% RSLogix 500 project I2P-Job-12 Part 2 Duncan_Sutton.RSS, saved by version 10.00.00.00 %
PROJECT "ML01A"    % processor: Bul.1763 MicroLogix 1100 Series B %

PROGRAM FILES
  LAD 2   9 rungs

DATA FILES
  O0 OUTPUT  4 elements
  I1 INPUT  6 elements
  S2 STATUS  66 elements
  B3 BINARY  1 elements
  T4 TIMER  1 elements
  C5 COUNTER  1 elements
  R6 CONTROL  1 elements
  N7 INTEGER  1 elements
  F8 FLOAT  1 elements

LADDER 2
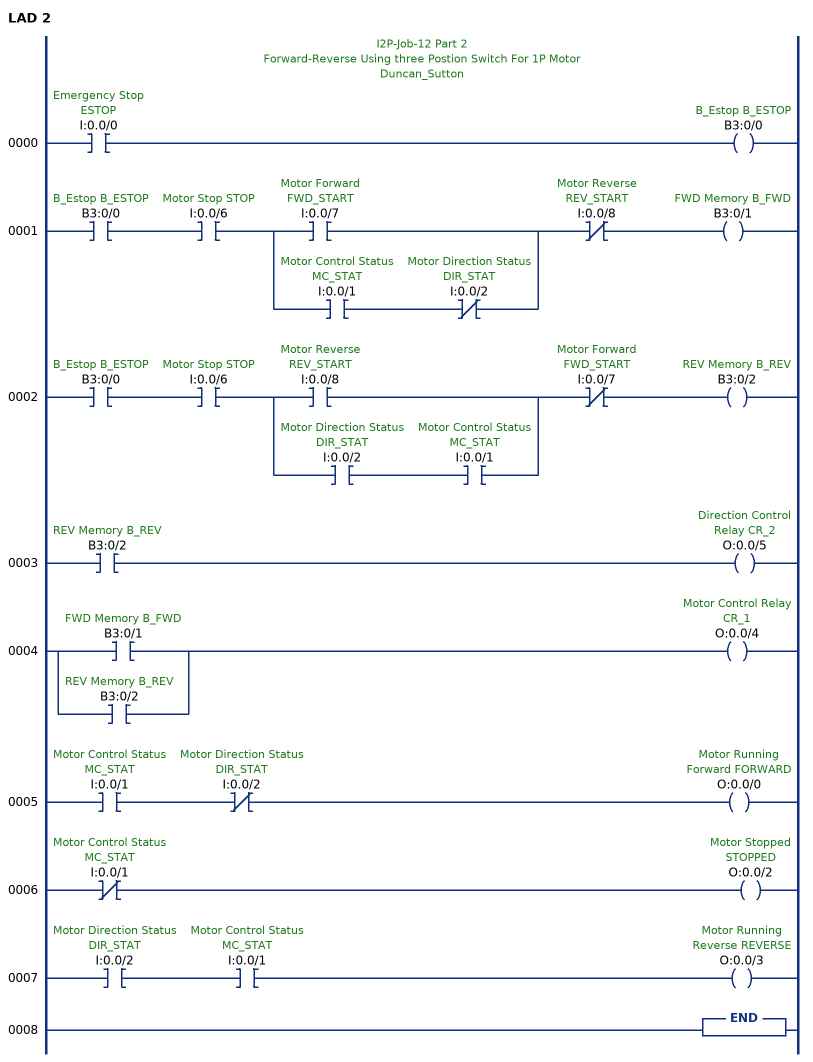
% Rung: 0 %
% I2P-Job-12 Part 2
% Forward-Reverse Using three Postion Switch For 1P Motor
% Duncan_Sutton %
SOR XIC I:0.0/0 OTE B3:0/0 EOR
%   I:0.0/0  ESTOP  "Emergency Stop" %
%   B3:0/0  B_ESTOP  "B_Estop" %
% Rung: 1 %
SOR XIC B3:0/0 XIC I:0.0/6 BST XIC I:0.0/7 NXB XIC I:0.0/1 XIO I:0.0/2 BND XIO I:0.0/8 OTE B3:0/1 EOR
%   B3:0/0  B_ESTOP  "B_Estop" %
%   I:0.0/6  STOP  "Motor Stop" %
%   I:0.0/7  FWD_START  "Motor Forward" %
%   I:0.0/1  MC_STAT  "Motor Control Status" %
%   I:0.0/2  DIR_STAT  "Motor Direction Status" %
%   I:0.0/8  REV_START  "Motor Reverse" %
%   B3:0/1  B_FWD  "FWD Memory" %
% Rung: 2 %
SOR XIC B3:0/0 XIC I:0.0/6 BST XIC I:0.0/8 NXB XIC I:0.0/2 XIC I:0.0/1 BND XIO I:0.0/7 OTE B3:0/2 EOR
%   B3:0/0  B_ESTOP  "B_Estop" %
%   I:0.0/6  STOP  "Motor Stop" %
%   I:0.0/8  REV_START  "Motor Reverse" %
%   I:0.0/2  DIR_STAT  "Motor Direction Status" %
%   I:0.0/1  MC_STAT  "Motor Control Status" %
%   I:0.0/7  FWD_START  "Motor Forward" %
%   B3:0/2  B_REV  "REV Memory" %
% Rung: 3 %
SOR XIC B3:0/2 OTE O:0.0/5 EOR
%   B3:0/2  B_REV  "REV Memory" %
%   O:0.0/5  CR_2  "Direction Control Relay" %
% Rung: 4 %
SOR BST XIC B3:0/1 NXB XIC B3:0/2 BND OTE O:0.0/4 EOR
%   B3:0/1  B_FWD  "FWD Memory" %
%   B3:0/2  B_REV  "REV Memory" %
%   O:0.0/4  CR_1  "Motor Control Relay" %
% Rung: 5 %
SOR XIC I:0.0/1 XIO I:0.0/2 OTE O:0.0/0 EOR
%   I:0.0/1  MC_STAT  "Motor Control Status" %
%   I:0.0/2  DIR_STAT  "Motor Direction Status" %
%   O:0.0/0  FORWARD  "Motor Running Forward" %
% Rung: 6 %
SOR XIO I:0.0/1 OTE O:0.0/2 EOR
%   I:0.0/1  MC_STAT  "Motor Control Status" %
%   O:0.0/2  STOPPED  "Motor Stopped" %
% Rung: 7 %
SOR XIC I:0.0/2 XIC I:0.0/1 OTE O:0.0/3 EOR
%   I:0.0/2  DIR_STAT  "Motor Direction Status" %
%   I:0.0/1  MC_STAT  "Motor Control Status" %
%   O:0.0/3  REVERSE  "Motor Running Reverse" %
% Rung: 8 %
SOR END EOR

OTHER DOCUMENTED ADDRESSES
  I:0.0/3  FWD  "Direction"
  I:0.0/4  REV  "Direction"
  I:0.0/5  2PSS_PA  "2 Poistion Selector Switch Position A"
  O:0.0/1  FORCE_WAIT  "Motor Forced Wait Time"
  T4:0  MTR_STOP
  TT  "TOF/1 Timer"

DATA TABLE (non-zero values as saved)
DATA T4
% .PRE .ACC %
% T4:0 % 800 0
